FUNCTION SetupHardware : BOOL
VAR
	iCardboardSlot : Cardboard;
	iCornerGuardSlot : CornerGuard;
	
	i : INT;
END_VAR

FOR iCardboardSlot:=1 TO Cardboard.size-1 BY 1 DO
	skidA22Left.setSlot(i := iCardboardSlot, material := TO_STRING(iCardboardSlot), error => );
	skidA22Right.setSlot(i := iCardboardSlot, material := TO_STRING(iCardboardSlot), error => );
END_FOR

//--------------------------------------------------

FOR iCornerGuardSlot:=1 TO CornerGuard.size-1 BY 1 DO
	magazineA22Left.setSlot(i := iCornerGuardSlot, material := TO_STRING(iCornerGuardSlot), error => );
	magazineA22Right.setSlot(i := iCornerGuardSlot, material := TO_STRING(iCornerGuardSlot), error => );
END_FOR

//--------------------------------------------------

FOR i:=1 TO GVL.maxQueue BY 1 DO
	{warning disable C0195}
	magazineA22Left.setOccupancy(i := i, occupancy := IntegerBitAccess( robot3.inputs[3], i-1) );
	skidA22Left.setOccupancy(i := i, occupancy := IntegerBitAccess( robot3.inputs[4], i-1) );
	
	magazineA22Right.setOccupancy(i := i, occupancy := IntegerBitAccess( robot4.inputs[3], i-1) );
	skidA22Right.setOccupancy(i := i, occupancy := IntegerBitAccess( robot4.inputs[4], i-1) );
	{warning restore C0195}
END_FOR

//--------------------------------------------------

verticalDriveA22Left.bEnable := 
verticalDriveA22Right.bEnable := 
horizontalDriveA22Left.bEnable := 
horizontalDriveA22Right.bEnable := 
pistonA22Bottom.bEnable := 
TRUE;

END_FUNCTION

(* stored: Version 1.1.0.1, ProductVersion 3.1.4024.11
   POU SetupHardware: Id {ad70243f-26d6-4655-b24b-2a994d19bc18}, SpecialFunc None *)
